// TIA Portal V15.1 export
// export: Created 2024-05-17T05:38:10.3162537Z, ExportSetting WithDefaults, DisplayName Totally Integrated Automation Portal, DisplayVersion V15.1 Update 5, DisplayName TIA Portal Openness, DisplayVersion V15.1 Update 5, DisplayName SINAMICS Startdrive Advanced, DisplayVersion V15.1, DisplayName G130, G150, S120, S150, SINAMICS MV, S210, DisplayVersion V15.1, DisplayName G110M, G120, G120C, G120D, G120P, DisplayVersion V15.1, DisplayName STEP 7 Professional, DisplayVersion V15.1 Update 5, DisplayName STEP 7 Safety, DisplayVersion V15.1, DisplayName WinCC Professional, DisplayVersion V15.1 Update 5, DisplayName SIMATIC Visualization Architect, DisplayVersion V15.1
DATA_BLOCK "_209000NCP01PhoneAlarmReqString"   // DB1026
{ S7_Optimized_Access := 'FALSE' }
AUTHOR : VCC
FAMILY : Function
VERSION : 0.1
// stored: AutoNumber false, DBAccessibleFromOPCUA true, InstanceOfName LPhoneAlarmReqString, InstanceOfType FB
"LPhoneAlarmReqString"
   // VAR_INPUT
   //    I_PhoneAlarmReq1 { ExternalAccessible := 'False'; ExternalVisible := 'False'; ExternalWritable := 'False'} : Bool;
   //    I_PhoneAlarmReq2 { ExternalAccessible := 'False'; ExternalVisible := 'False'; ExternalWritable := 'False'} : Bool;
   //    I_PhoneAlarmReq3 { ExternalAccessible := 'False'; ExternalVisible := 'False'; ExternalWritable := 'False'} : Bool;
   //    I_PhoneAlarmReq4 { ExternalAccessible := 'False'; ExternalVisible := 'False'; ExternalWritable := 'False'} : Bool;
   //    I_PhoneAlarmReq5 { ExternalAccessible := 'False'; ExternalVisible := 'False'; ExternalWritable := 'False'} : Bool;
   //    I_PhoneAlarmReq6 { ExternalAccessible := 'False'; ExternalVisible := 'False'; ExternalWritable := 'False'} : Bool;
   //    I_PhoneAlarmReq7 { ExternalAccessible := 'False'; ExternalVisible := 'False'; ExternalWritable := 'False'} : Bool;
   //    I_PhoneAlarmReq8 { ExternalAccessible := 'False'; ExternalVisible := 'False'; ExternalWritable := 'False'} : Bool;
   //    I_PhoneAlarmReq9 { ExternalAccessible := 'False'; ExternalVisible := 'False'; ExternalWritable := 'False'} : Bool;
   //    I_PhoneAlarmReq10 { ExternalAccessible := 'False'; ExternalVisible := 'False'; ExternalWritable := 'False'} : Bool;
   //    I_PhoneAlarmReq11 { ExternalAccessible := 'False'; ExternalVisible := 'False'; ExternalWritable := 'False'} : Bool;
   //    I_PhoneAlarmReq12 { ExternalAccessible := 'False'; ExternalVisible := 'False'; ExternalWritable := 'False'} : Bool;
   //    I_PhoneAlarmReq13 { ExternalAccessible := 'False'; ExternalVisible := 'False'; ExternalWritable := 'False'} : Bool;
   //    I_PhoneAlarmReq14 { ExternalAccessible := 'False'; ExternalVisible := 'False'; ExternalWritable := 'False'} : Bool;
   //    I_PhoneAlarmReq15 { ExternalAccessible := 'False'; ExternalVisible := 'False'; ExternalWritable := 'False'} : Bool;
   //    I_PhoneAlarmReq16 { ExternalAccessible := 'False'; ExternalVisible := 'False'; ExternalWritable := 'False'} : Bool;
   //    C_MessageType1 { ExternalAccessible := 'False'; ExternalVisible := 'False'; ExternalWritable := 'False'} : String[20];
   //    C_Message1 { ExternalAccessible := 'False'; ExternalVisible := 'False'; ExternalWritable := 'False'} : String[120];
   //    C_MessageType2 { ExternalAccessible := 'False'; ExternalVisible := 'False'; ExternalWritable := 'False'} : String[20];
   //    C_Message2 { ExternalAccessible := 'False'; ExternalVisible := 'False'; ExternalWritable := 'False'} : String[120];
   //    C_MessageType3 { ExternalAccessible := 'False'; ExternalVisible := 'False'; ExternalWritable := 'False'} : String[20];
   //    C_Message3 { ExternalAccessible := 'False'; ExternalVisible := 'False'; ExternalWritable := 'False'} : String[120];
   //    C_MessageType4 { ExternalAccessible := 'False'; ExternalVisible := 'False'; ExternalWritable := 'False'} : String[20];
   //    C_Message4 { ExternalAccessible := 'False'; ExternalVisible := 'False'; ExternalWritable := 'False'} : String[120];
   //    C_MessageType5 { ExternalAccessible := 'False'; ExternalVisible := 'False'; ExternalWritable := 'False'} : String[20];
   //    C_Message5 { ExternalAccessible := 'False'; ExternalVisible := 'False'; ExternalWritable := 'False'} : String[120];
   //    C_MessageType6 { ExternalAccessible := 'False'; ExternalVisible := 'False'; ExternalWritable := 'False'} : String[20];
   //    C_Message6 { ExternalAccessible := 'False'; ExternalVisible := 'False'; ExternalWritable := 'False'} : String[120];
   //    C_MessageType7 { ExternalAccessible := 'False'; ExternalVisible := 'False'; ExternalWritable := 'False'} : String[20];
   //    C_Message7 { ExternalAccessible := 'False'; ExternalVisible := 'False'; ExternalWritable := 'False'} : String[120];
   //    C_MessageType8 { ExternalAccessible := 'False'; ExternalVisible := 'False'; ExternalWritable := 'False'} : String[20];
   //    C_Message8 { ExternalAccessible := 'False'; ExternalVisible := 'False'; ExternalWritable := 'False'} : String[120];
   //    C_MessageType9 { ExternalAccessible := 'False'; ExternalVisible := 'False'; ExternalWritable := 'False'} : String[20];
   //    C_Message9 { ExternalAccessible := 'False'; ExternalVisible := 'False'; ExternalWritable := 'False'} : String[120];
   //    C_MessageType10 { ExternalAccessible := 'False'; ExternalVisible := 'False'; ExternalWritable := 'False'} : String[20];
   //    C_Message10 { ExternalAccessible := 'False'; ExternalVisible := 'False'; ExternalWritable := 'False'} : String[120];
   //    C_MessageType11 { ExternalAccessible := 'False'; ExternalVisible := 'False'; ExternalWritable := 'False'} : String[20];
   //    C_Message11 { ExternalAccessible := 'False'; ExternalVisible := 'False'; ExternalWritable := 'False'} : String[120];
   //    C_MessageType12 { ExternalAccessible := 'False'; ExternalVisible := 'False'; ExternalWritable := 'False'} : String[20];
   //    C_Message12 { ExternalAccessible := 'False'; ExternalVisible := 'False'; ExternalWritable := 'False'} : String[120];
   //    C_MessageType13 { ExternalAccessible := 'False'; ExternalVisible := 'False'; ExternalWritable := 'False'} : String[20];
   //    C_Message13 { ExternalAccessible := 'False'; ExternalVisible := 'False'; ExternalWritable := 'False'} : String[120];
   //    C_MessageType14 { ExternalAccessible := 'False'; ExternalVisible := 'False'; ExternalWritable := 'False'} : String[20];
   //    C_Message14 { ExternalAccessible := 'False'; ExternalVisible := 'False'; ExternalWritable := 'False'} : String[120];
   //    C_MessageType15 { ExternalAccessible := 'False'; ExternalVisible := 'False'; ExternalWritable := 'False'} : String[20];
   //    C_Message15 { ExternalAccessible := 'False'; ExternalVisible := 'False'; ExternalWritable := 'False'} : String[120];
   //    C_MessageType16 { ExternalAccessible := 'False'; ExternalVisible := 'False'; ExternalWritable := 'False'} : String[20];
   //    C_Message16 { ExternalAccessible := 'False'; ExternalVisible := 'False'; ExternalWritable := 'False'} : String[120];
   //    C_VDCommRecvDB { ExternalAccessible := 'False'; ExternalVisible := 'False'; ExternalWritable := 'False'} : DB_ANY;
   //    C_VDCommSendDB { ExternalAccessible := 'False'; ExternalVisible := 'False'; ExternalWritable := 'False'} : DB_ANY;
   //    C_LocalRecvDB { ExternalAccessible := 'False'; ExternalVisible := 'False'; ExternalWritable := 'False'} : DB_ANY;
   //    C_LocalSendDB { ExternalAccessible := 'False'; ExternalVisible := 'False'; ExternalWritable := 'False'} : DB_ANY;
   //    C_SubSystem { ExternalAccessible := 'False'; ExternalVisible := 'False'; ExternalWritable := 'False'} : Int;
   //    C_FilterMessage1 { ExternalAccessible := 'False'; ExternalVisible := 'False'; ExternalWritable := 'False'} : Time;
   //    C_FilterMessage2 { ExternalAccessible := 'False'; ExternalVisible := 'False'; ExternalWritable := 'False'} : Time;
   //    C_FilterMessage3 { ExternalAccessible := 'False'; ExternalVisible := 'False'; ExternalWritable := 'False'} : Time;
   //    C_FilterMessage4 { ExternalAccessible := 'False'; ExternalVisible := 'False'; ExternalWritable := 'False'} : Time;
   //    C_FilterMessage5 { ExternalAccessible := 'False'; ExternalVisible := 'False'; ExternalWritable := 'False'} : Time;
   //    C_FilterMessage6 { ExternalAccessible := 'False'; ExternalVisible := 'False'; ExternalWritable := 'False'} : Time;
   //    C_FilterMessage7 { ExternalAccessible := 'False'; ExternalVisible := 'False'; ExternalWritable := 'False'} : Time;
   //    C_FilterMessage8 { ExternalAccessible := 'False'; ExternalVisible := 'False'; ExternalWritable := 'False'} : Time;
   //    C_FilterMessage9 { ExternalAccessible := 'False'; ExternalVisible := 'False'; ExternalWritable := 'False'} : Time;
   //    C_FilterMessage10 { ExternalAccessible := 'False'; ExternalVisible := 'False'; ExternalWritable := 'False'} : Time;
   //    C_FilterMessage11 { ExternalAccessible := 'False'; ExternalVisible := 'False'; ExternalWritable := 'False'} : Time;
   //    C_FilterMessage12 { ExternalAccessible := 'False'; ExternalVisible := 'False'; ExternalWritable := 'False'} : Time;
   //    C_FilterMessage13 { ExternalAccessible := 'False'; ExternalVisible := 'False'; ExternalWritable := 'False'} : Time;
   //    C_FilterMessage14 { ExternalAccessible := 'False'; ExternalVisible := 'False'; ExternalWritable := 'False'} : Time;
   //    C_FilterMessage15 { ExternalAccessible := 'False'; ExternalVisible := 'False'; ExternalWritable := 'False'} : Time;
   //    C_FilterMessage16 { ExternalAccessible := 'False'; ExternalVisible := 'False'; ExternalWritable := 'False'} : Time;
   // END_VAR
   // VAR_IN_OUT
   //    IO_VD : "VDComm";
   //    H_HMI : "H_HMI";
   //    H_PhoneAlarmReqString : "H_PhoneAlarmReqString";
   // END_VAR
   // VAR
   //    ReqPhoneAlarm { ExternalAccessible := 'False'; ExternalVisible := 'False'; ExternalWritable := 'False'} : Array[1..16] of Bool;
   //    VDReqPhoneAlarm { ExternalAccessible := 'False'; ExternalVisible := 'False'; ExternalWritable := 'False'} : Array[1..16] of Bool;
   //    Done { ExternalAccessible := 'False'; ExternalVisible := 'False'; ExternalWritable := 'False'} : Array[1..16] of Bool;
   //    StnEdge { ExternalAccessible := 'False'; ExternalVisible := 'False'; ExternalWritable := 'False'} : Array[1..16] of Bool;
   //    SendDoneToVD { ExternalAccessible := 'False'; ExternalVisible := 'False'; ExternalWritable := 'False'} : Bool;
   //    SendVD { ExternalAccessible := 'False'; ExternalVisible := 'False'; ExternalWritable := 'False'} : Bool;
   //    PhoneAlarmReqActiveStn1 { ExternalAccessible := 'False'; ExternalVisible := 'False'; ExternalWritable := 'False'} : Bool;
   //    PhoneAlarmReqActiveStn2 { ExternalAccessible := 'False'; ExternalVisible := 'False'; ExternalWritable := 'False'} : Bool;
   //    PhoneAlarmReqActiveStn3 { ExternalAccessible := 'False'; ExternalVisible := 'False'; ExternalWritable := 'False'} : Bool;
   //    PhoneAlarmReqActiveStn4 { ExternalAccessible := 'False'; ExternalVisible := 'False'; ExternalWritable := 'False'} : Bool;
   //    PhoneAlarmReqActiveStn5 { ExternalAccessible := 'False'; ExternalVisible := 'False'; ExternalWritable := 'False'} : Bool;
   //    PhoneAlarmReqActiveStn6 { ExternalAccessible := 'False'; ExternalVisible := 'False'; ExternalWritable := 'False'} : Bool;
   //    PhoneAlarmReqActiveStn7 { ExternalAccessible := 'False'; ExternalVisible := 'False'; ExternalWritable := 'False'} : Bool;
   //    PhoneAlarmReqActiveStn8 { ExternalAccessible := 'False'; ExternalVisible := 'False'; ExternalWritable := 'False'} : Bool;
   //    PhoneAlarmReqActiveStn9 { ExternalAccessible := 'False'; ExternalVisible := 'False'; ExternalWritable := 'False'} : Bool;
   //    PhoneAlarmReqActiveStn10 { ExternalAccessible := 'False'; ExternalVisible := 'False'; ExternalWritable := 'False'} : Bool;
   //    PhoneAlarmReqActiveStn11 { ExternalAccessible := 'False'; ExternalVisible := 'False'; ExternalWritable := 'False'} : Bool;
   //    PhoneAlarmReqActiveStn12 { ExternalAccessible := 'False'; ExternalVisible := 'False'; ExternalWritable := 'False'} : Bool;
   //    PhoneAlarmReqActiveStn13 { ExternalAccessible := 'False'; ExternalVisible := 'False'; ExternalWritable := 'False'} : Bool;
   //    PhoneAlarmReqActiveStn14 { ExternalAccessible := 'False'; ExternalVisible := 'False'; ExternalWritable := 'False'} : Bool;
   //    PhoneAlarmReqActiveStn15 { ExternalAccessible := 'False'; ExternalVisible := 'False'; ExternalWritable := 'False'} : Bool;
   //    PhoneAlarmReqActiveStn16 { ExternalAccessible := 'False'; ExternalVisible := 'False'; ExternalWritable := 'False'} : Bool;
   //    VDMessage { ExternalAccessible := 'False'; ExternalVisible := 'False'; ExternalWritable := 'False'} : Struct
   //       VDMessageType { ExternalAccessible := 'False'; ExternalVisible := 'False'; ExternalWritable := 'False'} : Array[0..19] of Byte;
   //       VDMessage { ExternalAccessible := 'False'; ExternalVisible := 'False'; ExternalWritable := 'False'} : Array[0..119] of Byte;
   //    END_STRUCT;
   //    _VDComSubSystem { ExternalAccessible := 'False'; ExternalVisible := 'False'; ExternalWritable := 'False'; S7_SetPoint := 'True'} : "LVDComSubSystemS7-1500";
   //    Edge { ExternalAccessible := 'False'; ExternalVisible := 'False'; ExternalWritable := 'False'} : Array[0..15] of Bool;
   //    InitDone { ExternalAccessible := 'False'; ExternalVisible := 'False'; ExternalWritable := 'False'} : Array[1..32] of Bool;
   //    InitDoneEdge { ExternalAccessible := 'False'; ExternalVisible := 'False'; ExternalWritable := 'False'} : Array[1..32] of Bool;
   //    MessageType { ExternalAccessible := 'False'; ExternalVisible := 'False'; ExternalWritable := 'False'} : Int;
   //    MessageLength { ExternalAccessible := 'False'; ExternalVisible := 'False'; ExternalWritable := 'False'} : Word;
   //    _Filter1 { ExternalAccessible := 'False'; ExternalVisible := 'False'; ExternalWritable := 'False'; S7_SetPoint := 'True'} : TON_TIME;
   //    _Filter2 { ExternalAccessible := 'False'; ExternalVisible := 'False'; ExternalWritable := 'False'; S7_SetPoint := 'True'} : TON_TIME;
   //    _Filter3 { ExternalAccessible := 'False'; ExternalVisible := 'False'; ExternalWritable := 'False'; S7_SetPoint := 'True'} : TON_TIME;
   //    _Filter4 { ExternalAccessible := 'False'; ExternalVisible := 'False'; ExternalWritable := 'False'; S7_SetPoint := 'True'} : TON_TIME;
   //    _Filter5 { ExternalAccessible := 'False'; ExternalVisible := 'False'; ExternalWritable := 'False'; S7_SetPoint := 'True'} : TON_TIME;
   //    _Filter6 { ExternalAccessible := 'False'; ExternalVisible := 'False'; ExternalWritable := 'False'; S7_SetPoint := 'True'} : TON_TIME;
   //    _Filter7 { ExternalAccessible := 'False'; ExternalVisible := 'False'; ExternalWritable := 'False'; S7_SetPoint := 'True'} : TON_TIME;
   //    _Filter8 { ExternalAccessible := 'False'; ExternalVisible := 'False'; ExternalWritable := 'False'; S7_SetPoint := 'True'} : TON_TIME;
   //    _Filter9 { ExternalAccessible := 'False'; ExternalVisible := 'False'; ExternalWritable := 'False'; S7_SetPoint := 'True'} : TON_TIME;
   //    _Filter10 { ExternalAccessible := 'False'; ExternalVisible := 'False'; ExternalWritable := 'False'; S7_SetPoint := 'True'} : TON_TIME;
   //    _Filter11 { ExternalAccessible := 'False'; ExternalVisible := 'False'; ExternalWritable := 'False'; S7_SetPoint := 'True'} : TON_TIME;
   //    _Filter12 { ExternalAccessible := 'False'; ExternalVisible := 'False'; ExternalWritable := 'False'; S7_SetPoint := 'True'} : TON_TIME;
   //    _Filter13 { ExternalAccessible := 'False'; ExternalVisible := 'False'; ExternalWritable := 'False'; S7_SetPoint := 'True'} : TON_TIME;
   //    _Filter14 { ExternalAccessible := 'False'; ExternalVisible := 'False'; ExternalWritable := 'False'; S7_SetPoint := 'True'} : TON_TIME;
   //    _Filter15 { ExternalAccessible := 'False'; ExternalVisible := 'False'; ExternalWritable := 'False'; S7_SetPoint := 'True'} : TON_TIME;
   //    _Filter16 { ExternalAccessible := 'False'; ExternalVisible := 'False'; ExternalWritable := 'False'; S7_SetPoint := 'True'} : TON_TIME;
   //    SendToVDTimeOut { ExternalAccessible := 'False'; ExternalVisible := 'False'; ExternalWritable := 'False'; S7_SetPoint := 'True'} : TON_TIME;
   //    ResetVDComm { ExternalAccessible := 'False'; ExternalVisible := 'False'; ExternalWritable := 'False'} : Bool;
   //    VDMessageTypeTemp { ExternalAccessible := 'False'; ExternalVisible := 'False'; ExternalWritable := 'False'} : String[20];
   //    VDMessageTemp { ExternalAccessible := 'False'; ExternalVisible := 'False'; ExternalWritable := 'False'} : String[120];
   //    VDMessageTypeSerialzePos { ExternalAccessible := 'False'; ExternalVisible := 'False'; ExternalWritable := 'False'} : DInt;
   //    VDMessageSerialzePos { ExternalAccessible := 'False'; ExternalVisible := 'False'; ExternalWritable := 'False'} : DInt;
   //    VDMessageTypeTempArray { ExternalAccessible := 'False'; ExternalVisible := 'False'; ExternalWritable := 'False'} : Array[0..21] of Byte;
   //    VDMessageTempArray { ExternalAccessible := 'False'; ExternalVisible := 'False'; ExternalWritable := 'False'} : Array[0..121] of Byte;
   // END_VAR
BEGIN
END_DATA_BLOCK
